FUNCTION_BLOCK EL3314
VAR
	_io : EL3xx4_Data;
	{attribute addProperty Name "WcState"}
	_wcState : WcStateInputToggle;
	{attribute addProperty Name "Info data"}
	_infoData : InfoDataAds;
END_VAR

PROPERTY IO : REFERENCE TO EL3xx4_Data
GET
IO REF= _io;
END_GET
END_PROPERTY

PROPERTY WcState : REFERENCE TO WcStateInputToggle
GET
WcState REF= _wcState;
END_GET
END_PROPERTY

END_FUNCTION_BLOCK

(* stored: Version 1.1.0.1, ProductVersion 3.1.4024.9
   POU EL3314: Id {7d105fba-b587-0ff3-1bc1-b17056da5416}, SpecialFunc None
   Property IO: Id {5e5a3be7-4e11-01e5-27e7-6079ab2fb124}
   Get Get: Id {147083f6-5d35-015b-01b1-89e9f42a65a6}
   Property WcState: Id {179da0c8-d658-0bab-338d-5ccedf2477f8}
   Get Get: Id {faf4375b-10bb-00b2-0958-1da33d786018} *)
